LIN {X 0,Y 65.601,Z 469.654,A -85,B 0,C 180,E1 -29395.769,E2 -29395.769} C_VEL
LIN {X 0,Y 60.85,Z 474.556,A -85,B 0,C 180,E1 -29402.479,E2 -29402.479} C_VEL
LIN {X 0,Y 56.182,Z 479.346,A -85,B 0,C 180,E1 -29411.771,E2 -29411.771} C_VEL
LIN {X 0,Y 52.961,Z 483.057,A -85,B 0,C 180,E1 -29422.369,E2 -29422.369} C_VEL
LIN {X 0,Y 51.792,Z 484.99,A -85,B 0,C 180,E1 -29429.994,E2 -29429.994} C_VEL
LIN {X 0,Y 51.666,Z 486.463,A -85,B 0,C 180,E1 -29437.812,E2 -29437.812} C_VEL
LIN {X 0,Y 53.686,Z 488.228,A -85,B 0,C 180,E1 -29453.118,E2 -29453.118} C_VEL
LIN {X 0,Y 57.553,Z 488.496,A -85,B 0,C 180,E1 -29464.256,E2 -29464.256} C_VEL
LIN {X 0,Y 62.31,Z 487.958,A -85,B 0,C 180,E1 -29472.584,E2 -29472.584} C_VEL
LIN {X 0,Y 70.975,Z 485.778,A -85,B 0,C 180,E1 -29482.382,E2 -29482.382} C_VEL
LIN {X 0,Y 75.17,Z 484.316,A -85,B 0,C 180,E1 -29485.903,E2 -29485.903} C_VEL
LIN {X 0,Y 77.381,Z 483.364,A -85,B 0,C 180,E1 -29488.293,E2 -29488.293} C_VEL
LIN {X 0,Y 82.987,Z 480.221,A -85,B 0,C 180,E1 -29496.791,E2 -29496.791} C_VEL
LIN {X 0,Y 85.618,Z 478.798,A -85,B 0,C 180,E1 -29498.583,E2 -29498.583} C_VEL
LIN {X 0,Y 85.944,Z 478.627,A -85,B 0,C 180,E1 -29498.731,E2 -29498.731} C_VEL
LIN {X 0,Y 87.515,Z 477.564,A -85,B 0,C 180,E1 -29501.262,E2 -29501.262} C_VEL
LIN {X 0,Y 89.272,Z 476.143,A -85,B 0,C 180,E1 -29506.338,E2 -29506.338} C_VEL
LIN {X 0,Y 90.619,Z 475.119,A -85,B 0,C 180,E1 -29511.076,E2 -29511.076} C_VEL
LIN {X 0,Y 91.958,Z 474.377,A -85,B 0,C 180,E1 -29515.616,E2 -29515.616} C_VEL
LIN {X 0,Y 93.418,Z 473.819,A -85,B 0,C 180,E1 -29519.999,E2 -29519.999} C_VEL
LIN {X 0,Y 92.704,Z 475.012,A -85,B 0,C 180,E1 -29524.347,E2 -29524.347} C_VEL
LIN {X 0,Y 91.664,Z 476.769,A -85,B 0,C 180,E1 -29528.82,E2 -29528.82} C_VEL
LIN {X 0,Y 90.259,Z 479.089,A -85,B 0,C 180,E1 -29533.508,E2 -29533.508} C_VEL
LIN {X 0,Y 89.564,Z 480.163,A -85,B 0,C 180,E1 -29535.469,E2 -29535.469} C_VEL
LIN {X 0,Y 88.455,Z 481.556,A -85,B 0,C 180,E1 -29537.564,E2 -29537.564} C_VEL
LIN {X 0,Y 82.824,Z 485.515,A -85,B 0,C 180,E1 -29541.038,E2 -29541.038} C_VEL
LIN {X 0,Y 77.246,Z 488.878,A -85,B 0,C 180,E1 -29544.528,E2 -29544.528} C_VEL
LIN {X 0,Y 71.565,Z 491.702,A -85,B 0,C 180,E1 -29547.899,E2 -29547.899} C_VEL
LIN {X 0,Y 62.585,Z 495.268,A -85,B 0,C 180,E1 -29554.156,E2 -29554.156} C_VEL
LIN {X 0,Y 55.827,Z 497.39,A -85,B 0,C 180,E1 -29560.954,E2 -29560.954} C_VEL
LIN {X 0,Y 47.942,Z 499.211,A -85,B 0,C 180,E1 -29574.107,E2 -29574.107} C_VEL
LIN {X 0,Y 43.667,Z 499.462,A -85,B 0,C 180,E1 -29591.23,E2 -29591.23} C_VEL
LIN {X 0,Y 43.218,Z 499.03,A -85,B 0,C 180,E1 -29600.648,E2 -29600.648} C_VEL
LIN {X 0,Y 43.428,Z 498.152,A -85,B 0,C 180,E1 -29610.007,E2 -29610.007} C_VEL
LIN {X 0,Y 42.93,Z 496.298,A -85,B 0,C 180,E1 -29620.824,E2 -29620.824} C_VEL
LIN {X 0,Y 45.077,Z 492.064,A -85,B 0,C 180,E1 -29637.895,E2 -29637.895} C_VEL
LIN {X 0,Y 49.415,Z 487.409,A -85,B 0,C 180,E1 -29649.8,E2 -29649.8} C_VEL
LIN {X 0,Y 55.549,Z 481.534,A -85,B 0,C 180,E1 -29659.394,E2 -29659.394} C_VEL
LIN {X 0,Y 62.099,Z 473.906,A -85,B 0,C 180,E1 -29668.09,E2 -29668.09} C_VEL
LIN {X 0,Y 68.207,Z 466.081,A -85,B 0,C 180,E1 -29674.378,E2 -29674.378} C_VEL
LIN {X 0,Y 73.484,Z 458.4,A -85,B 0,C 180,E1 -29679.16,E2 -29679.16} C_VEL
LIN {X 0,Y 75.708,Z 454.561,A -85,B 0,C 180,E1 -29681.451,E2 -29681.451} C_VEL
LIN {X 0,Y 76.606,Z 449.848,A -85,B 0,C 180,E1 -29686.742,E2 -29686.742} C_VEL
LIN {X 0,Y 76.967,Z 447.652,A -85,B 0,C 180,E1 -29689.478,E2 -29689.478} C_VEL
LIN {X 0,Y 77.033,Z 446.051,A -85,B 0,C 180,E1 -29692.136,E2 -29692.136} C_VEL
LIN {X 0,Y 76.944,Z 444.877,A -85,B 0,C 180,E1 -29694.761,E2 -29694.761} C_VEL
LIN {X 0,Y 76.642,Z 443.336,A -85,B 0,C 180,E1 -29700.001,E2 -29700.001} C_VEL
LIN {X 0,Y 75.844,Z 443.161,A -85,B 0,C 180,E1 -29706.791,E2 -29706.791} C_VEL
LIN {X 0,Y 75.646,Z 443.361,A -85,B 0,C 180,E1 -29710.71,E2 -29710.71} C_VEL
LIN {X 0,Y 75.321,Z 444.496,A -85,B 0,C 180,E1 -29716.257,E2 -29716.257} C_VEL
LIN {X 0,Y 75.131,Z 446.224,A -85,B 0,C 180,E1 -29721.975,E2 -29721.975} C_VEL
LIN {X 0,Y 74.873,Z 448.895,A -85,B 0,C 180,E1 -29727.992,E2 -29727.992} C_VEL
LIN {X 0,Y 74.433,Z 452.55,A -85,B 0,C 180,E1 -29734.51,E2 -29734.51} C_VEL
LIN {X 0,Y 73.635,Z 456.398,A -85,B 0,C 180,E1 -29740.215,E2 -29740.215} C_VEL
LIN {X 0,Y 65.85,Z 465.004,A -85,B 0,C 180,E1 -29746.068,E2 -29746.068} C_VEL
LIN {X 0,Y 58.814,Z 471.877,A -85,B 0,C 180,E1 -29753.305,E2 -29753.305} C_VEL
LIN {X 0,Y 52.865,Z 477.384,A -85,B 0,C 180,E1 -29762.264,E2 -29762.264} C_VEL
LIN {X 0,Y 48.126,Z 481.757,A -85,B 0,C 180,E1 -29773.012,E2 -29773.012} C_VEL
LIN {X 0,Y 45.946,Z 484.085,A -85,B 0,C 180,E1 -29781.195,E2 -29781.195} C_VEL
LIN {X 0,Y 44.719,Z 485.991,A -85,B 0,C 180,E1 -29789.993,E2 -29789.993} C_VEL
LIN {X 0,Y 44.667,Z 487.418,A -85,B 0,C 180,E1 -29799.046,E2 -29799.046} C_VEL
LIN {X 0,Y 47.224,Z 489.143,A -85,B 0,C 180,E1 -29816.51,E2 -29816.51} C_VEL
LIN {X 0,Y 49.827,Z 489.442,A -85,B 0,C 180,E1 -29824.339,E2 -29824.339} C_VEL
LIN {X 0,Y 57.254,Z 488.784,A -85,B 0,C 180,E1 -29837.427,E2 -29837.427} C_VEL
LIN {X 0,Y 61.824,Z 487.872,A -85,B 0,C 180,E1 -29842.718,E2 -29842.718} C_VEL
LIN {X 0,Y 70.825,Z 485.264,A -85,B 0,C 180,E1 -29850.253,E2 -29850.253} C_VEL
LIN {X 0,Y 80.651,Z 481.257,A -85,B 0,C 180,E1 -29856.193,E2 -29856.193} C_VEL
LIN {X 0,Y 85.618,Z 478.798,A -85,B 0,C 180,E1 -29858.583,E2 -29858.583} C_VEL
LIN {X 0,Y 87.199,Z 477.904,A -85,B 0,C 180,E1 -29859.829,E2 -29859.829} C_VEL
LIN {X 0,Y 88.245,Z 477.168,A -85,B 0,C 180,E1 -29862.018,E2 -29862.018} C_VEL
LIN {X 0,Y 88.413,Z 476.834,A -85,B 0,C 180,E1 -29865.134,E2 -29865.134} C_VEL
LIN {X 0,Y 87.978,Z 476.912,A -85,B 0,C 180,E1 -29867.67,E2 -29867.67} C_VEL
LIN {X 0,Y 86.44,Z 477.766,A -85,B 0,C 180,E1 -29876.817,E2 -29876.817} C_VEL
LIN {X 0,Y 87.125,Z 477.66,A -85,B 0,C 180,E1 -29879.84,E2 -29879.84} C_VEL
LIN {X 0,Y 86.364,Z 478.882,A -85,B 0,C 180,E1 -29884.667,E2 -29884.667} C_VEL
LIN {X 0,Y 85.008,Z 480.755,A -85,B 0,C 180,E1 -29889.516,E2 -29889.516} C_VEL
LIN {X 0,Y 84.124,Z 481.886,A -85,B 0,C 180,E1 -29892.054,E2 -29892.054} C_VEL
LIN {X 0,Y 82.433,Z 483.544,A -85,B 0,C 180,E1 -29894.818,E2 -29894.818} C_VEL
LIN {X 0,Y 74.471,Z 488.166,A -85,B 0,C 180,E1 -29899.327,E2 -29899.327} C_VEL
LIN {X 0,Y 68.503,Z 490.989,A -85,B 0,C 180,E1 -29902.591,E2 -29902.591} C_VEL
LIN {X 0,Y 58.226,Z 494.711,A -85,B 0,C 180,E1 -29908.867,E2 -29908.867} C_VEL
LIN {X 0,Y 51.421,Z 496.582,A -85,B 0,C 180,E1 -29914.92,E2 -29914.92} C_VEL
LIN {X 0,Y 46.539,Z 497.659,A -85,B 0,C 180,E1 -29920.978,E2 -29920.978} C_VEL
LIN {X 0,Y 42.358,Z 498.342,A -85,B 0,C 180,E1 -29928.428,E2 -29928.428} C_VEL
LIN {X 0,Y 36.981,Z 498.545,A -85,B 0,C 180,E1 -29947.67,E2 -29947.67} C_VEL
LIN {X 0,Y 36.202,Z 498.092,A -85,B 0,C 180,E1 -29958.814,E2 -29958.814} C_VEL
LIN {X 0,Y 36.281,Z 497.182,A -85,B 0,C 180,E1 -29970.008,E2 -29970.008} C_VEL
LIN {X 0,Y 36.101,Z 494.71,A -85,B 0,C 180,E1 -29986.405,E2 -29986.405} C_VEL
LIN {X 0,Y 38.883,Z 491.003,A -85,B 0,C 180,E1 -30002.846,E2 -30002.846} C_VEL
LIN {X 0,Y 44.14,Z 486.293,A -85,B 0,C 180,E1 -30015.775,E2 -30015.775} C_VEL
LIN {X 0,Y 51.063,Z 480.311,A -85,B 0,C 180,E1 -30025.68,E2 -30025.68} C_VEL
LIN {X 0,Y 58.495,Z 472.586,A -85,B 0,C 180,E1 -30034.315,E2 -30034.315} C_VEL
LIN {X 0,Y 65.25,Z 464.674,A -85,B 0,C 180,E1 -30040.417,E2 -30040.417} C_VEL
LIN {X 0,Y 70.264,Z 457.979,A -85,B 0,C 180,E1 -30044.517,E2 -30044.517} C_VEL
LIN {X 0,Y 70.91,Z 456.653,A -85,B 0,C 180,E1 -30045.665,E2 -30045.665} C_VEL
LIN {X 0,Y 72.164,Z 452.356,A -85,B 0,C 180,E1 -30051.319,E2 -30051.319} C_VEL
LIN {X 0,Y 72.37,Z 450.721,A -85,B 0,C 180,E1 -30054.428,E2 -30054.428} C_VEL
LIN {X 0,Y 72.225,Z 449.025,A -85,B 0,C 180,E1 -30060.001,E2 -30060.001} C_VEL
LIN {X 0,Y 71.512,Z 448.758,A -85,B 0,C 180,E1 -30066.518,E2 -30066.518} C_VEL
LIN {X 0,Y 71.106,Z 449.144,A -85,B 0,C 180,E1 -30071.402,E2 -30071.402} C_VEL
LIN {X 0,Y 70.594,Z 450.359,A -85,B 0,C 180,E1 -30077.379,E2 -30077.379} C_VEL
LIN {X 0,Y 70.173,Z 452.313,A -85,B 0,C 180,E1 -30083.618,E2 -30083.618} C_VEL
LIN {X 0,Y 69.398,Z 455.42,A -85,B 0,C 180,E1 -30090.423,E2 -30090.423} C_VEL
LIN {X 0,Y 68.681,Z 457.933,A -85,B 0,C 180,E1 -30095.045,E2 -30095.045} C_VEL
LIN {X 0,Y 67.894,Z 459.286,A -85,B 0,C 180,E1 -30096.649,E2 -30096.649} C_VEL
LIN {X 0,Y 59.65,Z 467.451,A -85,B 0,C 180,E1 -30102.569,E2 -30102.569} C_VEL
LIN {X 0,Y 53.339,Z 473.033,A -85,B 0,C 180,E1 -30108.784,E2 -30108.784} C_VEL
LIN {X 0,Y 46.729,Z 478.487,A -85,B 0,C 180,E1 -30118.23,E2 -30118.23} C_VEL
LIN {X 0,Y 41.42,Z 482.808,A -85,B 0,C 180,E1 -30130.155,E2 -30130.155} C_VEL
LIN {X 0,Y 38.959,Z 485.114,A -85,B 0,C 180,E1 -30139.6,E2 -30139.6} C_VEL
LIN {X 0,Y 37.645,Z 486.981,A -85,B 0,C 180,E1 -30149.992,E2 -30149.992} C_VEL
LIN {X 0,Y 37.678,Z 488.375,A -85,B 0,C 180,E1 -30160.742,E2 -30160.742} C_VEL
LIN {X 0,Y 41.061,Z 490.067,A -85,B 0,C 180,E1 -30181.148,E2 -30181.148} C_VEL
LIN {X 0,Y 44.14,Z 490.317,A -85,B 0,C 180,E1 -30189.551,E2 -30189.551} C_VEL
LIN {X 0,Y 52.69,Z 489.609,A -85,B 0,C 180,E1 -30203.149,E2 -30203.149} C_VEL
LIN {X 0,Y 57.779,Z 488.674,A -85,B 0,C 180,E1 -30208.361,E2 -30208.361} C_VEL
LIN {X 0,Y 67.082,Z 486.163,A -85,B 0,C 180,E1 -30215.222,E2 -30215.222} C_VEL
LIN {X 0,Y 78.039,Z 481.936,A -85,B 0,C 180,E1 -30221.003,E2 -30221.003} C_VEL
LIN {X 0,Y 81.083,Z 480.541,A -85,B 0,C 180,E1 -30222.436,E2 -30222.436} C_VEL
LIN {X 0,Y 82.285,Z 479.805,A -85,B 0,C 180,E1 -30225.152,E2 -30225.152} C_VEL
LIN {X 0,Y 83.988,Z 478.827,A -85,B 0,C 180,E1 -30230.365,E2 -30230.365} C_VEL
LIN {X 0,Y 85.583,Z 478.137,A -85,B 0,C 180,E1 -30235.289,E2 -30235.289} C_VEL
LIN {X 0,Y 87.125,Z 477.66,A -85,B 0,C 180,E1 -30239.84,E2 -30239.84} C_VEL
LIN {X 0,Y 87.262,Z 477.818,A -85,B 0,C 180,E1 -30241.485,E2 -30241.485} C_VEL
LIN {X 0,Y 86.413,Z 478.641,A -85,B 0,C 180,E1 -30243.468,E2 -30243.468} C_VEL
LIN {X 0,Y 84.099,Z 480.385,A -85,B 0,C 180,E1 -30245.954,E2 -30245.954} C_VEL
LIN {X 0,Y 80.267,Z 482.937,A -85,B 0,C 180,E1 -30248.727,E2 -30248.727} C_VEL
LIN {X 0,Y 76.228,Z 485.381,A -85,B 0,C 180,E1 -30251.52,E2 -30251.52} C_VEL
LIN {X 0,Y 75.122,Z 486.061,A -85,B 0,C 180,E1 -30252.357,E2 -30252.357} C_VEL
LIN {X 0,Y 69.211,Z 488.918,A -85,B 0,C 180,E1 -30255.291,E2 -30255.291} C_VEL
LIN {X 0,Y 62.894,Z 491.436,A -85,B 0,C 180,E1 -30258.244,E2 -30258.244} C_VEL
LIN {X 0,Y 53.581,Z 494.344,A -85,B 0,C 180,E1 -30263.354,E2 -30263.354} C_VEL
LIN {X 0,Y 42.207,Z 496.83,A -85,B 0,C 180,E1 -30273.65,E2 -30273.65} C_VEL
LIN {X 0,Y 33.286,Z 497.729,A -85,B 0,C 180,E1 -30290.708,E2 -30290.708} C_VEL
LIN {X 0,Y 29.224,Z 497.153,A -85,B 0,C 180,E1 -30316.095,E2 -30316.095} C_VEL
LIN {X 0,Y 29.132,Z 496.201,A -85,B 0,C 180,E1 -30330.01,E2 -30330.01} C_VEL
LIN {X 0,Y 29.364,Z 493.593,A -85,B 0,C 180,E1 -30351.05,E2 -30351.05} C_VEL
LIN {X 0,Y 33.078,Z 489.933,A -85,B 0,C 180,E1 -30369.61,E2 -30369.61} C_VEL
LIN {X 0,Y 39.479,Z 485.167,A -85,B 0,C 180,E1 -30383.246,E2 -30383.246} C_VEL
LIN {X 0,Y 45.977,Z 480.211,A -85,B 0,C 180,E1 -30391.528,E2 -30391.528} C_VEL
LIN {X 0,Y 54.2,Z 472.707,A -85,B 0,C 180,E1 -30400.083,E2 -30400.083} C_VEL
LIN {X 0,Y 62.622,Z 463.776,A -85,B 0,C 180,E1 -30406.67,E2 -30406.67} C_VEL
LIN {X 0,Y 65.451,Z 460.396,A -85,B 0,C 180,E1 -30408.711,E2 -30408.711} C_VEL
LIN {X 0,Y 66.161,Z 459.256,A -85,B 0,C 180,E1 -30409.787,E2 -30409.787} C_VEL
LIN {X 0,Y 67.293,Z 456.5,A -85,B 0,C 180,E1 -30414.006,E2 -30414.006} C_VEL
LIN {X 0,Y 67.451,Z 455.319,A -85,B 0,C 180,E1 -30417.015,E2 -30417.015} C_VEL
LIN {X 0,Y 67.483,Z 454.48,A -85,B 0,C 180,E1 -30420.001,E2 -30420.001} C_VEL
LIN {X 0,Y 66.9,Z 454.123,A -85,B 0,C 180,E1 -30426.032,E2 -30426.032} C_VEL
LIN {X 0,Y 66.19,Z 454.696,A -85,B 0,C 180,E1 -30432.262,E2 -30432.262} C_VEL
LIN {X 0,Y 65.793,Z 455.335,A -85,B 0,C 180,E1 -30435.958,E2 -30435.958} C_VEL
LIN {X 0,Y 65.109,Z 457.028,A -85,B 0,C 180,E1 -30442.199,E2 -30442.199} C_VEL
LIN {X 0,Y 64.046,Z 459.596,A -85,B 0,C 180,E1 -30448.604,E2 -30448.604} C_VEL
LIN {X 0,Y 63.546,Z 460.719,A -85,B 0,C 180,E1 -30450.995,E2 -30450.995} C_VEL
LIN {X 0,Y 62.452,Z 462.046,A -85,B 0,C 180,E1 -30452.426,E2 -30452.426} C_VEL
LIN {X 0,Y 53.733,Z 469.882,A -85,B 0,C 180,E1 -30458.291,E2 -30458.291} C_VEL
LIN {X 0,Y 45.732,Z 476.134,A -85,B 0,C 180,E1 -30466.238,E2 -30466.238} C_VEL
LIN {X 0,Y 38.687,Z 481.145,A -85,B 0,C 180,E1 -30476.967,E2 -30476.967} C_VEL
LIN {X 0,Y 33.315,Z 485.056,A -85,B 0,C 180,E1 -30491.544,E2 -30491.544} C_VEL
LIN {X 0,Y 30.567,Z 487.962,A -85,B 0,C 180,E1 -30509.99,E2 -30509.99} C_VEL
LIN {X 0,Y 30.738,Z 489.333,A -85,B 0,C 180,E1 -30523.207,E2 -30523.207} C_VEL
LIN {X 0,Y 35.082,Z 490.969,A -85,B 0,C 180,E1 -30546.931,E2 -30546.931} C_VEL
LIN {X 0,Y 38.901,Z 491.189,A -85,B 0,C 180,E1 -30556.263,E2 -30556.263} C_VEL
LIN {X 0,Y 48.751,Z 490.432,A -85,B 0,C 180,E1 -30569.866,E2 -30569.866} C_VEL
LIN {X 0,Y 54.374,Z 489.475,A -85,B 0,C 180,E1 -30574.779,E2 -30574.779} C_VEL
LIN {X 0,Y 63.909,Z 487.058,A -85,B 0,C 180,E1 -30580.735,E2 -30580.735} C_VEL
LIN {X 0,Y 75.282,Z 482.928,A -85,B 0,C 180,E1 -30585.855,E2 -30585.855} C_VEL
LIN {X 0,Y 77.018,Z 482.211,A -85,B 0,C 180,E1 -30589.483,E2 -30589.483} C_VEL
LIN {X 0,Y 78.958,Z 481.503,A -85,B 0,C 180,E1 -30594.892,E2 -30594.892} C_VEL
LIN {X 0,Y 80.722,Z 481.142,A -85,B 0,C 180,E1 -30599.999,E2 -30599.999} C_VEL
LIN {X 0,Y 79.673,Z 482.457,A -85,B 0,C 180,E1 -30605.06,E2 -30605.06} C_VEL
LIN {X 0,Y 78.327,Z 483.936,A -85,B 0,C 180,E1 -30609.277,E2 -30609.277} C_VEL
LIN {X 0,Y 77.769,Z 484.448,A -85,B 0,C 180,E1 -30610.412,E2 -30610.412} C_VEL
LIN {X 0,Y 76.228,Z 485.381,A -85,B 0,C 180,E1 -30611.52,E2 -30611.52} C_VEL
LIN {X 0,Y 73.34,Z 486.936,A -85,B 0,C 180,E1 -30613.1,E2 -30613.1} C_VEL
LIN {X 0,Y 68.165,Z 489.105,A -85,B 0,C 180,E1 -30614.543,E2 -30614.543} C_VEL
LIN {X 0,Y 58.505,Z 492.003,A -85,B 0,C 180,E1 -30615.536,E2 -30615.536} C_VEL
LIN {X 0,Y 50.519,Z 493.795,A -85,B 0,C 180,E1 -30616.8,E2 -30616.8} C_VEL
LIN {X 0,Y 46.75,Z 494.533,A -85,B 0,C 180,E1 -30618.466,E2 -30618.466} C_VEL
LIN {X 0,Y 38.714,Z 495.992,A -85,B 0,C 180,E1 -30624.832,E2 -30624.832} C_VEL
LIN {X 0,Y 28.131,Z 496.836,A -85,B 0,C 180,E1 -30641.469,E2 -30641.469} C_VEL
LIN {X 0,Y 22.371,Z 496.215,A -85,B 0,C 180,E1 -30671.704,E2 -30671.704} C_VEL
LIN {X 0,Y 21.983,Z 495.215,A -85,B 0,C 180,E1 -30690.013,E2 -30690.013} C_VEL
LIN {X 0,Y 22.824,Z 492.561,A -85,B 0,C 180,E1 -30717.523,E2 -30717.523} C_VEL
LIN {X 0,Y 27.915,Z 488.849,A -85,B 0,C 180,E1 -30739.067,E2 -30739.067} C_VEL
LIN {X 0,Y 35.661,Z 484.03,A -85,B 0,C 180,E1 -30752.498,E2 -30752.498} C_VEL
LIN {X 0,Y 41.279,Z 480.234,A -85,B 0,C 180,E1 -30758.515,E2 -30758.515} C_VEL
LIN {X 0,Y 50.546,Z 472.776,A -85,B 0,C 180,E1 -30766.753,E2 -30766.753} C_VEL
LIN {X 0,Y 59.638,Z 464.111,A -85,B 0,C 180,E1 -30772.736,E2 -30772.736} C_VEL
LIN {X 0,Y 60.644,Z 463.029,A -85,B 0,C 180,E1 -30773.347,E2 -30773.347} C_VEL
LIN {X 0,Y 61.834,Z 461.442,A -85,B 0,C 180,E1 -30775.111,E2 -30775.111} C_VEL
LIN {X 0,Y 62.227,Z 460.637,A -85,B 0,C 180,E1 -30776.764,E2 -30776.764} C_VEL
LIN {X 0,Y 62.446,Z 459.663,A -85,B 0,C 180,E1 -30780.001,E2 -30780.001} C_VEL
LIN {X 0,Y 61.816,Z 459.314,A -85,B 0,C 180,E1 -30786.53,E2 -30786.53} C_VEL
LIN {X 0,Y 60.933,Z 459.94,A -85,B 0,C 180,E1 -30793.339,E2 -30793.339} C_VEL
LIN {X 0,Y 59.864,Z 461.557,A -85,B 0,C 180,E1 -30800.623,E2 -30800.623} C_VEL
LIN {X 0,Y 58.616,Z 463.601,A -85,B 0,C 180,E1 -30806.466,E2 -30806.466} C_VEL
LIN {X 0,Y 55.84,Z 466.091,A -85,B 0,C 180,E1 -30808.223,E2 -30808.223} C_VEL
LIN {X 0,Y 46.664,Z 473.297,A -85,B 0,C 180,E1 -30814.06,E2 -30814.06} C_VEL
LIN {X 0,Y 38.146,Z 479.068,A -85,B 0,C 180,E1 -30822.515,E2 -30822.515} C_VEL
LIN {X 0,Y 30.67,Z 483.643,A -85,B 0,C 180,E1 -30835.038,E2 -30835.038} C_VEL
LIN {X 0,Y 25.155,Z 487.168,A -85,B 0,C 180,E1 -30853.764,E2 -30853.764} C_VEL
LIN {X 0,Y 23.489,Z 488.941,A -85,B 0,C 180,E1 -30869.988,E2 -30869.988} C_VEL
LIN {X 0,Y 23.874,Z 490.292,A -85,B 0,C 180,E1 -30887.108,E2 -30887.108} C_VEL
LIN {X 0,Y 29.692,Z 491.879,A -85,B 0,C 180,E1 -30915.229,E2 -30915.229} C_VEL
LIN {X 0,Y 39.745,Z 491.85,A -85,B 0,C 180,E1 -30932.13,E2 -30932.13} C_VEL
LIN {X 0,Y 51.737,Z 490.266,A -85,B 0,C 180,E1 -30941.951,E2 -30941.951} C_VEL
LIN {X 0,Y 61.311,Z 487.975,A -85,B 0,C 180,E1 -30946.745,E2 -30946.745} C_VEL
LIN {X 0,Y 67.939,Z 485.858,A -85,B 0,C 180,E1 -30949.315,E2 -30949.315} C_VEL
LIN {X 0,Y 71.016,Z 484.817,A -85,B 0,C 180,E1 -30951.715,E2 -30951.715} C_VEL
LIN {X 0,Y 72.049,Z 484.542,A -85,B 0,C 180,E1 -30954.401,E2 -30954.401} C_VEL
LIN {X 0,Y 74.045,Z 484.244,A -85,B 0,C 180,E1 -30959.999,E2 -30959.999} C_VEL
LIN {X 0,Y 72.652,Z 485.635,A -85,B 0,C 180,E1 -30965.55,E2 -30965.55} C_VEL
LIN {X 0,Y 70.934,Z 486.728,A -85,B 0,C 180,E1 -30967.819,E2 -30967.819} C_VEL
LIN {X 0,Y 64.338,Z 489.531,A -85,B 0,C 180,E1 -30970.57,E2 -30970.57} C_VEL
LIN {X 0,Y 57.712,Z 491.759,A -85,B 0,C 180,E1 -30973.06,E2 -30973.06} C_VEL
LIN {X 0,Y 46.75,Z 494.533,A -85,B 0,C 180,E1 -30978.466,E2 -30978.466} C_VEL
LIN {X 0,Y 41.335,Z 495.475,A -85,B 0,C 180,E1 -30981.311,E2 -30981.311} C_VEL
LIN {X 0,Y 31.808,Z 496.173,A -85,B 0,C 180,E1 -30985.549,E2 -30985.549} C_VEL
LIN {X 0,Y 22.649,Z 496.061,A -85,B 0,C 180,E1 -30993.634,E2 -30993.634} C_VEL
LIN {X 0,Y 18.343,Z 495.712,A -85,B 0,C 180,E1 -31004.964,E2 -31004.964} C_VEL
LIN {X 0,Y 15.747,Z 495.264,A -85,B 0,C 180,E1 -31023.514,E2 -31023.514} C_VEL
LIN {X 0,Y 14.831,Z 494.229,A -85,B 0,C 180,E1 -31050.02,E2 -31050.02} C_VEL
LIN {X 0,Y 16.791,Z 491.524,A -85,B 0,C 180,E1 -31088.912,E2 -31088.912} C_VEL
LIN {X 0,Y 23.835,Z 487.76,A -85,B 0,C 180,E1 -31112.228,E2 -31112.228} C_VEL
LIN {X 0,Y 32.968,Z 482.889,A -85,B 0,C 180,E1 -31123.627,E2 -31123.627} C_VEL
LIN {X 0,Y 38.574,Z 479.422,A -85,B 0,C 180,E1 -31128.209,E2 -31128.209} C_VEL
LIN {X 0,Y 47.676,Z 472.808,A -85,B 0,C 180,E1 -31134.347,E2 -31134.347} C_VEL
LIN {X 0,Y 56.241,Z 465.455,A -85,B 0,C 180,E1 -31138.799,E2 -31138.799} C_VEL
LIN {X 0,Y 57.025,Z 464.576,A -85,B 0,C 180,E1 -31140.002,E2 -31140.002} C_VEL
LIN {X 0,Y 56.557,Z 464.136,A -85,B 0,C 180,E1 -31146.172,E2 -31146.172} C_VEL
LIN {X 0,Y 55.139,Z 465.113,A -85,B 0,C 180,E1 -31154.771,E2 -31154.771} C_VEL
LIN {X 0,Y 54.666,Z 465.653,A -85,B 0,C 180,E1 -31157.795,E2 -31157.795} C_VEL
LIN {X 0,Y 52.871,Z 467.348,A -85,B 0,C 180,E1 -31161.475,E2 -31161.475} C_VEL
LIN {X 0,Y 43.123,Z 474.483,A -85,B 0,C 180,E1 -31166.299,E2 -31166.299} C_VEL
LIN {X 0,Y 33.786,Z 480.183,A -85,B 0,C 180,E1 -31173.675,E2 -31173.675} C_VEL
LIN {X 0,Y 25.216,Z 484.702,A -85,B 0,C 180,E1 -31185.815,E2 -31185.815} C_VEL
LIN {X 0,Y 18.462,Z 488.185,A -85,B 0,C 180,E1 -31207.607,E2 -31207.607} C_VEL
LIN {X 0,Y 17.211,Z 491.251,A -85,B 0,C 180,E1 -31254.082,E2 -31254.082} C_VEL
LIN {X 0,Y 23.939,Z 492.666,A -85,B 0,C 180,E1 -31284.039,E2 -31284.039} C_VEL
LIN {X 0,Y 30.82,Z 492.928,A -85,B 0,C 180,E1 -31295.779,E2 -31295.779} C_VEL
LIN {X 0,Y 43.377,Z 492.083,A -85,B 0,C 180,E1 -31306.411,E2 -31306.411} C_VEL
LIN {X 0,Y 49.988,Z 491.047,A -85,B 0,C 180,E1 -31309.753,E2 -31309.753} C_VEL
LIN {X 0,Y 59.482,Z 488.88,A -85,B 0,C 180,E1 -31313.213,E2 -31313.213} C_VEL
LIN {X 0,Y 63.547,Z 487.684,A -85,B 0,C 180,E1 -31314.428,E2 -31314.428} C_VEL
LIN {X 0,Y 66.131,Z 487.049,A -85,B 0,C 180,E1 -31317.325,E2 -31317.325} C_VEL
LIN {X 0,Y 67.114,Z 486.975,A -85,B 0,C 180,E1 -31319.999,E2 -31319.999} C_VEL
LIN {X 0,Y 66.649,Z 487.377,A -85,B 0,C 180,E1 -31321.912,E2 -31321.912} C_VEL
LIN {X 0,Y 63.403,Z 488.775,A -85,B 0,C 180,E1 -31324.023,E2 -31324.023} C_VEL
LIN {X 0,Y 56.526,Z 490.998,A -85,B 0,C 180,E1 -31325.976,E2 -31325.976} C_VEL
LIN {X 0,Y 42.912,Z 494.165,A -85,B 0,C 180,E1 -31330.72,E2 -31330.72} C_VEL
LIN {X 0,Y 29.917,Z 495.722,A -85,B 0,C 180,E1 -31340.033,E2 -31340.033} C_VEL
LIN {X 0,Y 18.98,Z 495.792,A -85,B 0,C 180,E1 -31362.242,E2 -31362.242} C_VEL
LIN {X 0,Y 18.343,Z 495.712,A -85,B 0,C 180,E1 -31364.964,E2 -31364.964} C_VEL
LIN {X 0,Y 16.043,Z 495.379,A -85,B 0,C 180,E1 -31375.469,E2 -31375.469} C_VEL
LIN {X 0,Y 13.744,Z 494.81,A -85,B 0,C 180,E1 -31387.592,E2 -31387.592} C_VEL
LIN {X 0,Y 10.991,Z 493.639,A -85,B 0,C 180,E1 -31411.916,E2 -31411.916} C_VEL
LIN {X 0,Y 11.802,Z 490.975,A -85,B 0,C 180,E1 -31463.298,E2 -31463.298} C_VEL
LIN {X 0,Y 15.835,Z 489.033,A -85,B 0,C 180,E1 -31481.136,E2 -31481.136} C_VEL
LIN {X 0,Y 17.512,Z 488.317,A -85,B 0,C 180,E1 -31484.46,E2 -31484.46} C_VEL
LIN {X 0,Y 28.246,Z 483.519,A -85,B 0,C 180,E1 -31494.523,E2 -31494.523} C_VEL
LIN {X 0,Y 35.167,Z 479.814,A -85,B 0,C 180,E1 -31497.971,E2 -31497.971} C_VEL
LIN {X 0,Y 45.74,Z 472.839,A -85,B 0,C 180,E1 -31502.748,E2 -31502.748} C_VEL
LIN {X 0,Y 49.329,Z 470.153,A -85,B 0,C 180,E1 -31504.134,E2 -31504.134} C_VEL
LIN {X 0,Y 51.084,Z 468.672,A -85,B 0,C 180,E1 -31505.412,E2 -31505.412} C_VEL
LIN {X 0,Y 49.55,Z 469.499,A -85,B 0,C 180,E1 -31513.851,E2 -31513.851} C_VEL
LIN {X 0,Y 45.6,Z 472.326,A -85,B 0,C 180,E1 -31515.553,E2 -31515.553} C_VEL
LIN {X 0,Y 37.134,Z 477.654,A -85,B 0,C 180,E1 -31518.839,E2 -31518.839} C_VEL
LIN {X 0,Y 27.164,Z 482.892,A -85,B 0,C 180,E1 -31525.078,E2 -31525.078} C_VEL
LIN {X 0,Y 17.676,Z 487.008,A -85,B 0,C 180,E1 -31537.299,E2 -31537.299} C_VEL
LIN {X 0,Y 12.215,Z 489.191,A -85,B 0,C 180,E1 -31554.845,E2 -31554.845} C_VEL
LIN {X 0,Y 11.111,Z 492.209,A -85,B 0,C 180,E1 -31629.201,E2 -31629.201} C_VEL
LIN {X 0,Y 19.961,Z 493.528,A -85,B 0,C 180,E1 -31659.38,E2 -31659.38} C_VEL
LIN {X 0,Y 28.643,Z 493.798,A -85,B 0,C 180,E1 -31668.897,E2 -31668.897} C_VEL
LIN {X 0,Y 42.274,Z 492.906,A -85,B 0,C 180,E1 -31675.845,E2 -31675.845} C_VEL
LIN {X 0,Y 49.222,Z 491.825,A -85,B 0,C 180,E1 -31677.949,E2 -31677.949} C_VEL
LIN {X 0,Y 49.191,Z 491.995,A -85,B 0,C 180,E1 -31679.757,E2 -31679.757} C_VEL
LIN {X 0,Y 42.171,Z 493.353,A -85,B 0,C 180,E1 -31681.139,E2 -31681.139} C_VEL
LIN {X 0,Y 28.277,Z 494.85,A -85,B 0,C 180,E1 -31686.295,E2 -31686.295} C_VEL
LIN {X 0,Y 15.135,Z 494.877,A -85,B 0,C 180,E1 -31701.817,E2 -31701.817} C_VEL
LIN {X 0,Y 9.69,Z 494.262,A -85,B 0,C 180,E1 -31726.482,E2 -31726.482} C_VEL
LIN {X 0,Y 7.684,Z 493.243,A -85,B 0,C 180,E1 -31770.038,E2 -31770.038} C_VEL
LIN {X 0,Y 12.075,Z 490.485,A -85,B 0,C 180,E1 -31830.865,E2 -31830.865} C_VEL
LIN {X 0,Y 17.512,Z 488.317,A -85,B 0,C 180,E1 -31844.46,E2 -31844.46} C_VEL
LIN {X 0,Y 17.168,Z 488.208,A -85,B 0,C 180,E1 -31847.599,E2 -31847.599} C_VEL
LIN {X 0,Y 15.165,Z 488.58,A -85,B 0,C 180,E1 -31851.934,E2 -31851.934} C_VEL
LIN {X 0,Y 12.057,Z 489.289,A -85,B 0,C 180,E1 -31856.959,E2 -31856.959} C_VEL
LIN {X 0,Y 3.309,Z 491.383,A -85,B 0,C 180,E1 -31892.303,E2 -31892.303} C_VEL
LIN {X 0,Y 3.49,Z 492.408,A -85,B 0,C 180,E1 -32006.157,E2 -32006.157} C_VEL
LIN {X 0,Y 7.183,Z 493.165,A -85,B 0,C 180,E1 -32027.863,E2 -32027.863} C_VEL
LIN {X 0,Y 7.025,Z 493.347,A -85,B 0,C 180,E1 -32038.728,E2 -32038.728} C_VEL
LIN {X 0,Y 0.545,Z 492.26,A -85,B 0,C 180,E1 -32130.535,E2 -32130.535} C_VEL
LIN {X 0,Y 10.627,Z 489.448,A -85,B 0,C 180,E1 -32227.036,E2 -32227.036} C_VEL
LIN {X 0,Y 21.338,Z 485.586,A -85,B 0,C 180,E1 -32228.76,E2 -32228.76} C_VEL
LIN {X 0,Y 28.5,Z 482.378,A -85,B 0,C 180,E1 -32229.405,E2 -32229.405} C_VEL
LIN {X 0,Y 18.01,Z 486.802,A -85,B 0,C 180,E1 -32232.614,E2 -32232.614} C_VEL
LIN {X 0,Y 7.609,Z 490.191,A -85,B 0,C 180,E1 -32242.435,E2 -32242.435} C_VEL
LIN {X 0,Y 3.49,Z 492.408,A -85,B 0,C 180,E1 -32366.157,E2 -32366.157} C_VEL
LIN {X 0,Y 4.865,Z 494.375,A -85,B 0,C 180,E1 -32378.635,E2 -32378.635} C_VEL
LIN {X 0,Y 4.865,Z 600,A -85,B 0,C 180,E1 -32378.635,E2 -32378.635} C_VEL
LIN {X 0,Y 4.865,Z 600,A -85,B 0,C 180,E1 -32378.635,E2 -32378.635}

QRS_NEXT_CUT()

QRS_NEXT()
QRS_HOME()

END
